// SIMATIC STEP 7 (V5.x) project Zaitsev_Lab2
// CPU: CPU 312
// station: Hardware
// station: SIMATIC 300(1)
// station: P_ADR_BUS
// program: S7 Program(1)

SYMBOL_TABLE
"Оператор"	I 0.0	BOOL
"Датчик движения"	I 0.1	BOOL
"Датчик разбития стекла"	I 0.2	BOOL
"Датчик дверей"	I 0.3	BOOL
"Сигнализация"	Q 0.0	BOOL
END_SYMBOL_TABLE

ORGANIZATION_BLOCK OB 1
TITLE = "Main Program Sweep (Cycle)"
VERSION : 0.1
VAR_TEMP
  OB1_EV_CLASS : BYTE ;	//Bits 0-3 = 1 (Coming event), Bits 4-7 = 1 (Event class 1)
  OB1_SCAN_1 : BYTE ;	//1 (Cold restart scan 1 of OB 1), 3 (Scan 2-n of OB 1)
  OB1_PRIORITY : BYTE ;	//Priority of OB Execution
  OB1_OB_NUMBR : BYTE ;	//1 (Organization block 1, OB1)
  OB1_RESERVED_1 : BYTE ;	//Reserved for system
  OB1_RESERVED_2 : BYTE ;	//Reserved for system
  OB1_PREV_CYCLE : INT ;	//Cycle time of previous OB1 scan (milliseconds)
  OB1_MIN_CYCLE : INT ;	//Minimum cycle time of OB1 (milliseconds)
  OB1_MAX_CYCLE : INT ;	//Maximum cycle time of OB1 (milliseconds)
  OB1_DATE_TIME : DATE_AND_TIME ;	//Date and time OB1 started
END_VAR
BEGIN
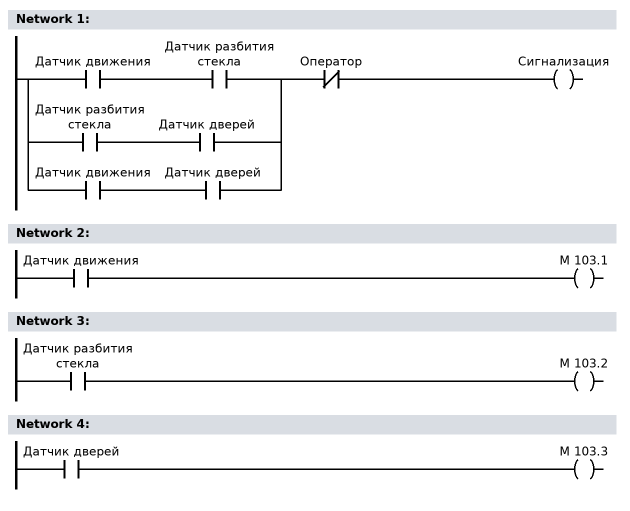
NETWORK
TITLE =
      A(;
      A     "Датчик движения";
      A     "Датчик разбития стекла";
      O;
      A     "Датчик разбития стекла";
      A     "Датчик дверей";
      O;
      A     "Датчик движения";
      A     "Датчик дверей";
      );
      AN    "Оператор";
      =     "Сигнализация";
NETWORK
TITLE =
      A     "Датчик движения";
      =     M 103.1;
NETWORK
TITLE =
      A     "Датчик разбития стекла";
      =     M 103.2;
NETWORK
TITLE =
      A     "Датчик дверей";
      =     M 103.3;
END_ORGANIZATION_BLOCK
